// TIA Portal V21 export
DATA_BLOCK "Sensore"   // DB30
{ S7_Optimized_Access := 'TRUE' }
// stored: MemoryReserve 100
   VAR
      S : Array[0.."K_NumSensore"] of "Std_Sensore";
   END_VAR
BEGIN
   S[0].In.Stato := FALSE;
   S[0].Prm.UnitàMisura.In.UmCode := 0;
   S[0].Prm.UnitàMisura.In.Valore := 0.0;
   S[0].Prm.UnitàMisura.Hmi.Converti := FALSE;
   S[0].Prm.UnitàMisura.Hmi.Calcola := FALSE;
   S[0].Prm.UnitàMisura.Dati.FattoreDiConversione := 0.0;
   S[0].Prm.UnitàMisura.Out.UmCode := 0;
   S[0].Prm.UnitàMisura.Out.Valore := 0.0;
   S[0].Hmi.ForzaPos := FALSE;
   S[0].Hmi.ForzaNeg := FALSE;
   S[0].Allarmi."A"[0..1].Abilitato := FALSE;
   S[0].Allarmi."A"[0..1].Stato := FALSE;
   S[0].Allarmi."A"[0..1].Silenziato := FALSE;
   S[0].Allarmi."A"[0..1].EnWarnHmi := FALSE;
   S[0].Allarmi."A"[0..1].EnCadutaCiclo := FALSE;
   S[0].Allarmi.WordHMI := 16#0000;
   S[0].Out.PresProd := FALSE;
   S[0].Out.Allarmi."A"[0..14].Abilitato := FALSE;
   S[0].Out.Allarmi."A"[0..14].Stato := FALSE;
   S[0].Out.Allarmi."A"[0..14].Silenziato := FALSE;
   S[0].Out.Allarmi."A"[0..14].EnWarnHmi := FALSE;
   S[0].Out.Allarmi."A"[0..14].EnCadutaCiclo := FALSE;
   S[0].Out.Allarmi.WordHMI := 16#0000;
   S[0].Rif_Inc.K_Zona := 0;
END_DATA_BLOCK
